(*
SPDX-FileCopyrightText: © 2026 Oleksandr Tiutyk <trofimich@gmail.com>
SPDX-License-Identifier: MIT
License: https://opensource.org/license/mit
*)

INTERFACE IEquatable EXTENDS __System.IQueryInterface

METHOD Equals : BOOL
VAR_IN_OUT CONSTANT
	otherObject : IEquatable;
END_VAR
END_METHOD

END_INTERFACE

(* stored: Version 1.1.0.1
   Itf IEquatable: Id {2e00bd23-1580-4f20-aa09-4d184e7e7028}
   Method Equals: Id {edad1141-8eff-463c-9dbe-f5b873637544} *)
